SUBAPPLICATION Uebung_011b3_PHYS (* Numeric Value Input SUB (PHYS) *)
  (* Standard: 61499-2; Description: Copyright (c) 2026 Meisterschulen am Ostbahnhof This program and the accompanying materials are made available under the terms of the Eclipse Public License 2.0 which is available at https://www.eclipse.org/legal/epl-2.0/ SPDX-License-Identifier: EPL-2.0 *)
  (* Version 1.0, 2026-04-24, Franz Höpfinger, Meisterschulen am Ostbahnhof, PHYS variant of Uebung_011b1 with REAL arithmetic *)
  PACKAGE Uebungen;
  IMPORT Uebungen::const::UT::DefaultPool_Numeric::InputNumber_I3_N;
  IMPORT Uebungen::const::UT::DefaultPool_Numeric::InputNumber_I4_N;
  IMPORT Uebungen::const::UT::DefaultPool_Numeric::OutputNumber_N3_N;
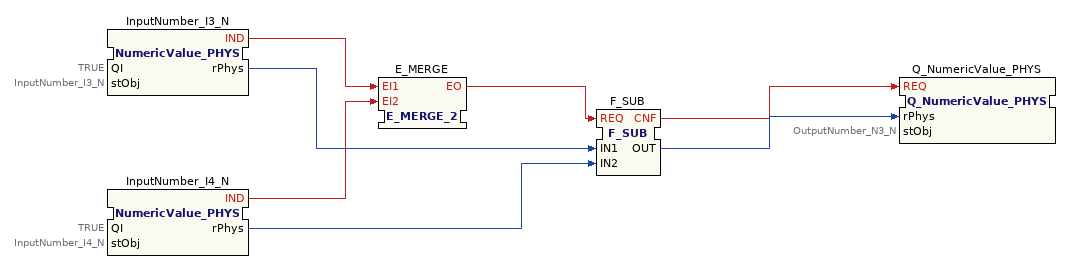
  FBS
    InputNumber_I3_N : isobus::UT::io::NumericValue::NumericValue_PHYS(QI := TRUE, stObj := InputNumber_I3_N);
    InputNumber_I4_N : isobus::UT::io::NumericValue::NumericValue_PHYS(QI := TRUE, stObj := InputNumber_I4_N);
    F_SUB : iec61131::arithmetic::F_SUB;
    Q_NumericValue_PHYS : isobus::UT::Q::Q_NumericValue_PHYS(stObj := OutputNumber_N3_N);
    E_MERGE : iec61499::events::E_MERGE_2;
  END_FBS
  EVENT_CONNECTIONS
    F_SUB.CNF TO Q_NumericValue_PHYS.REQ;
    E_MERGE.EO TO F_SUB.REQ;
    InputNumber_I3_N.IND TO E_MERGE.EI1;
    InputNumber_I4_N.IND TO E_MERGE.EI2;
  END_CONNECTIONS
  DATA_CONNECTIONS
    InputNumber_I3_N.rPhys TO F_SUB.IN1;
    F_SUB.OUT TO Q_NumericValue_PHYS.rPhys;
    InputNumber_I4_N.rPhys TO F_SUB.IN2;
  END_CONNECTIONS
END_SUBAPPLICATION
